// Mitsubishi GX Works2 project: Exercicio   PLC: Q03UDV

PROGRAM MAIN
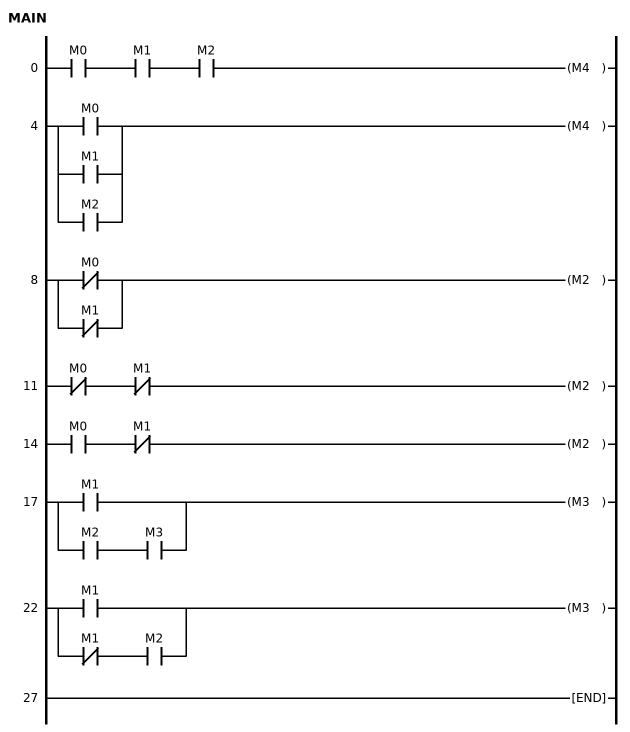
0     LD      M0
      AND     M1
      AND     M2
      OUT     M4
4     LD      M0
      OR      M1
      OR      M2
      OUT     M4
8     LDI     M0
      ORI     M1
      OUT     M2
11    LDI     M0
      ANI     M1
      OUT     M2
14    LD      M0
      ANI     M1
      OUT     M2
17    LD      M1
      LD      M2
      AND     M3
      ORB
      OUT     M3
22    LD      M1
      LDI     M1
      AND     M2
      ORB
      OUT     M3
27    END
END_PROGRAM
